TYPE T_OHM_Filename : STRING(44);
END_TYPE

(* stored: Version 1.1.0.1
   DUT T_OHM_Filename: Id {fb049b48-4f96-416a-950a-f2f0aac9e93f} *)
